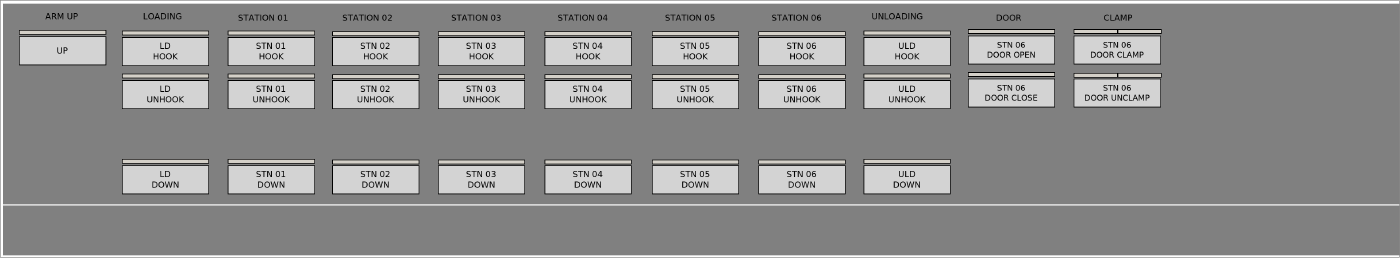
VISUALIZATION Popup_ArmControl  // 1918x354
    Rectangle (4,5 1914x275)
    Group (167,42 119x48)
        Rectangle (0,9 119x39), "LD HOOK", colour toggle: bArm1HorzLD1Hook_30
            toggle bArm1HorzLD1Hook_30
        RoundedRectangle (0,0 119x6), colour toggle: ARDSArmCtrl[1].AR3sbPositionCfm[2,1,8]
    Group (167,101 119x48)
        Rectangle (0,9 119x39), "LD UNHOOK", colour toggle: bArm1HorzLD1UnHook_30
            toggle bArm1HorzLD1UnHook_30
        RoundedRectangle (0,0 119x6), colour toggle: ARDSArmCtrl[1].AR3sbPositionCfm[2,1,7]
    Group (167,218 119x48)
        Rectangle (0,9 119x39), "LD DOWN", colour toggle: bArm1VertLD1Down_30
            toggle bArm1VertLD1Down_30
        RoundedRectangle (0,0 119x6), colour toggle: ARDSArmCtrl[1].AR3sbPositionCfm[2,1,6]
    Label (193,1 81x43), "LOADING"
    Group (312,42 119x48)
        Rectangle (0,9 119x39), "STN 01 HOOK", colour toggle: bArm1HorzStn1hook_30
            toggle bArm1HorzStn1hook_30
        RoundedRectangle (0,0 119x6), colour toggle: ARDSArmCtrl[1].AR3sbPositionCfm[1,1,8]
    Group (312,101 119x48)
        Rectangle (0,9 119x39), "STN 01 UNHOOK", colour toggle: bArm1HorzStn1Unhook_30
            toggle bArm1HorzStn1Unhook_30
        RoundedRectangle (0,0 119x6), colour toggle: ARDSArmCtrl[1].AR3sbPositionCfm[1,1,7]
    Group (312,218 119x48)
        Rectangle (0,9 119x39), "STN 01 DOWN", colour toggle: bArm1VertStn1Down_30
            toggle bArm1VertStn1Down_30
        RoundedRectangle (0,0 119x6), colour toggle: ARDSArmCtrl[1].AR3sbPositionCfm[1,1,6]
    Label (323,3 96x43), "STATION 01"
    Group (455,43 119x47)
        Rectangle (0,8 119x39), "STN 02 HOOK", colour toggle: bArm1HorzStn2hook_30
            toggle bArm1HorzStn2hook_30
        RoundedRectangle (0,0 119x6), colour toggle: ARDSArmCtrl[1].AR3sbPositionCfm[1,2,8]
    Group (455,102 119x47)
        Rectangle (0,8 119x39), "STN 02 UNHOOK", colour toggle: bArm1HorzStn2Unhook_30
            toggle bArm1HorzStn2Unhook_30
        RoundedRectangle (0,0 119x6), colour toggle: ARDSArmCtrl[1].AR3sbPositionCfm[1,2,7]
    Group (455,219 119x47)
        Rectangle (0,8 119x39), "STN 02 DOWN", colour toggle: bArm1VertStn2Down_30
            toggle bArm1VertStn2Down_30
        RoundedRectangle (0,0 119x6), colour toggle: ARDSArmCtrl[1].AR3sbPositionCfm[1,2,6]
    Label (466,3 96x43), "STATION 02"
    Group (600,43 119x47)
        Rectangle (0,8 119x39), "STN 03 HOOK", colour toggle: bArm1HorzStn3hook_30
            toggle bArm1HorzStn3hook_30
        RoundedRectangle (0,0 119x6), colour toggle: ARDSArmCtrl[1].AR3sbPositionCfm[1,3,8]
    Group (600,102 119x47)
        Rectangle (0,8 119x39), "STN 03 UNHOOK", colour toggle: bArm1HorzStn3Unhook_30
            toggle bArm1HorzStn3Unhook_30
        RoundedRectangle (0,0 119x6), colour toggle: ARDSArmCtrl[1].AR3sbPositionCfm[1,3,7]
    Group (600,219 119x47)
        Rectangle (0,8 119x39), "STN 03 DOWN", colour toggle: bArm1VertStn3Down_30
            toggle bArm1VertStn3Down_30
        RoundedRectangle (0,0 119x6), colour toggle: ARDSArmCtrl[1].AR3sbPositionCfm[1,3,6]
    Label (615,3 96x43), "STATION 03"
    Group (746,43 119x47)
        Rectangle (0,8 119x39), "STN 04 HOOK", colour toggle: bArm1HorzStn4hook_30
            toggle bArm1HorzStn4hook_30
        RoundedRectangle (0,0 119x6), colour toggle: ARDSArmCtrl[1].AR3sbPositionCfm[1,4,8]
    Group (746,102 119x47)
        Rectangle (0,8 119x39), "STN 04 UNHOOK", colour toggle: bArm1HorzStn4Unhook_30
            toggle bArm1HorzStn4Unhook_30
        RoundedRectangle (0,0 119x6), colour toggle: ARDSArmCtrl[1].AR3sbPositionCfm[1,4,7]
    Group (746,219 119x47)
        Rectangle (0,8 119x39), "STN 04 DOWN", colour toggle: bArm1VertStn4Down_30
            toggle bArm1VertStn4Down_30
        RoundedRectangle (0,0 119x6), colour toggle: ARDSArmCtrl[1].AR3sbPositionCfm[1,4,6]
    Label (761,3 96x43), "STATION 04"
    Group (893,43 119x47)
        Rectangle (0,8 119x39), "STN 05 HOOK", colour toggle: bArm1HorzStn5hook_30
            toggle bArm1HorzStn5hook_30
        RoundedRectangle (0,0 119x6), colour toggle: ARDSArmCtrl[1].AR3sbPositionCfm[1,5,8]
    Group (893,102 119x47)
        Rectangle (0,8 119x39), "STN 05 UNHOOK", colour toggle: bArm1HorzStn5Unhook_30
            toggle bArm1HorzStn5Unhook_30
        RoundedRectangle (0,0 119x6), colour toggle: ARDSArmCtrl[1].AR3sbPositionCfm[1,5,7]
    Group (893,219 119x47)
        Rectangle (0,8 119x39), "STN 05 DOWN", colour toggle: bArm1VertStn5Down_30
            toggle bArm1VertStn5Down_30
        RoundedRectangle (0,0 119x6), colour toggle: ARDSArmCtrl[1].AR3sbPositionCfm[1,5,6]
    Label (908,3 96x43), "STATION 05"
    Group (1039,43 119x47)
        Rectangle (0,8 119x39), "STN 06 HOOK", colour toggle: bArm1HorzStn6hook_30
            toggle .bArm1HorzStn6hook_30
        RoundedRectangle (0,0 119x6), colour toggle: ARDSArmCtrl[1].AR3sbPositionCfm[1,6,8]
    Group (1039,102 119x47)
        Rectangle (0,8 119x39), "STN 06 UNHOOK", colour toggle: bArm1HorzStn6Unhook_30
            toggle bArm1HorzStn6Unhook_30
        RoundedRectangle (0,0 119x6), colour toggle: ARDSArmCtrl[1].AR3sbPositionCfm[1,6,7]
    Group (1039,219 119x47)
        Rectangle (0,8 119x39), "STN 06 DOWN", colour toggle: bArm1VertStn6Down_30
            toggle bArm1VertStn6Down_30
        RoundedRectangle (0,0 119x6), colour toggle: ARDSArmCtrl[1].AR3sbPositionCfm[1,6,6]
    Label (1054,3 96x43), "STATION 06"
    Group (1183,42 119x48)
        Rectangle (0,9 119x39), "ULD HOOK", colour toggle: bArm1HorzULD1Hook_30
            toggle bArm1HorzULD1Hook_30
        RoundedRectangle (0,0 119x6), colour toggle: ARDSArmCtrl[1].AR3sbPositionCfm[3,1,8]
    Group (1183,101 119x48)
        Rectangle (0,9 119x39), "ULD UNHOOK", colour toggle: bArm1HorzULD1Unhook_30
            toggle bArm1HorzULD1Unhook_30
        RoundedRectangle (0,0 119x6), colour toggle: ARDSArmCtrl[1].AR3sbPositionCfm[3,1,7]
    Group (1183,218 119x48)
        Rectangle (0,9 119x39), "ULD DOWN", colour toggle: bArm1VertULD1Down_30
            toggle bArm1VertULD1Down_30
        RoundedRectangle (0,0 119x6), colour toggle: ARDSArmCtrl[1].AR3sbPositionCfm[3,1,6]
    Label (1191,1 102x43), "UNLOADING"
    Rectangle (4,282 1914x68)
    Group (26,41 119x48)
        Rectangle (0,9 119x39), "UP", colour toggle: bArm1VertLD1Up_30
            toggle bArm1VertLD1Up_30
        RoundedRectangle (0,0 119x6), colour toggle: ARDSArmCtrl[1].AR3sbPositionCfm[1,1,1]
    Label (59,-4 72x53), "ARM UP"
    Rectangle (1326,49 119x39), "STN 06 DOOR OPEN", colour toggle: bUldDoorOpen_15
        toggle bStn6DoorOpen_15
    RoundedRectangle (1326,40 119x6), colour toggle: ARbDI[eX12007_Stn06SlidingDoorRs_Open]
    Rectangle (1471,49 119x39), "STN 06 DOOR CLAMP", colour toggle: bUldDoorClose_15
        toggle ARwDO[eY12202_Stn06SlidingDoor_Clamp].15
    RoundedRectangle (1471,40 60x6), colour toggle: ARbDI[eX12100_Stn06SlidingDoorRs01_Clamp]
    Rectangle (1326,108 119x39), "STN 06 DOOR CLOSE", colour toggle: bUldConveyorOpen_15
        toggle bStn6DoorClose_15
    RoundedRectangle (1326,99 119x6), colour toggle: ARbDI[eX12008_Stn06SlidingDoorRs_Close]
    Rectangle (1471,108 119x39), "STN 06 DOOR UNCLAMP", colour toggle: bUldConveyorClose_15
        toggle ARwDO[eY12203_Stn06SlidingDoor_Unclamp].15
    Label (1334,3 96x43), "DOOR"
    Label (1484,3 96x43), "CLAMP"
    RoundedRectangle (1531,40 60x6), colour toggle: ARbDI[eX12102_Stn06SlidingDoorRs02_Clamp]
    RoundedRectangle (1531,100 60x6), colour toggle: ARbDI[eX12103_Stn06SlidingDoorRs02_Unclamp]
    RoundedRectangle (1471,100 60x6), colour toggle: ARbDI[eX12101_Stn06SlidingDoorRs01_Unclamp]
END_VISUALIZATION

(* stored: Version 1.1.0.1, ProductVersion 3.1.4024.12
   Visu Popup_ArmControl: Id {70995b9b-7dbe-4892-a237-17c9609b9cf8} *)
